FUNCTION_BLOCK RunCoordinator EXTENDS RunGroupNode
VAR_INPUT
	startProductionMode AT%I* : BOOL;
	startRegularCheckMode AT%I* : BOOL;
	//------------
	// link to HMI
	//------------
	purge AT%I* : BOOL ; 
	regularCheckAck AT%I* : BOOL;
END_VAR
VAR_OUTPUT
END_VAR
VAR
END_VAR

//Initialization sequences:
// 1. Group1 - two clamper and indexer (two clamper hold/unhold , the indexer turing 4 runs)
// 2. Group2 - SCARA1 and rack1,2 (pick to drop zone then homing and release rackes)
// 3. Group3 - SCARA2 and rack3,4

SUPER^();

CASE outputState OF
	//----------------------------
	//	Initializing :
	// 2. Off all I/O 
	// 1. SCARA & Clamper & Indexer
	//----------------------------	

	//------------------------------------------
	// Initialize - Group start (base procedure)
	//------------------------------------------
	eSpecialStates.GENERIC_GROUP_IDLE:
		//---------------------
		//	IDLE (Engineering mode): wait command / able to trigger individual process
		//---------------------
	//------------------------Working
	16#300:
		//----------------------------------
		//	Regular check mode
		//	1. Stand-along check SCARA1/SCARA2
		//	1. Bypass some stations then feed-in parts in Slot1 , then transit to AOI
		//  2. Prompt meesage/door interlock
		//----------------------------------
	16#500:
		//---------------------------
		//	Production mode
		//  1. Execute SCARA ASSEMBLE
		//	2. When purge command raise , coordinate stations to stop
		//---------------------------
		
END_CASE

END_FUNCTION_BLOCK

(* stored: Version 1.1.0.1, ProductVersion 3.1.4024.0
   POU RunCoordinator: Id {93db79ea-7610-40ae-89e3-5adae225f547}, SpecialFunc None *)
